FUNCTION_BLOCK PUBLIC FileSystemEntryCollection IMPLEMENTS I_FileSystemEntryCollection 
VAR
	entries : ARRAY[0..99] OF I_FileSystemEntry;
	currentIndex : INT := EMPTY;
	_nullEntry : NullEntry(Path:='');
END_VAR
VAR CONSTANT
	EMPTY : INT :=  -1;
END_VAR

METHOD Clear
VAR
	i : INT;
END_VAR
FOR i := 0 TO currentIndex DO
	entries[i] := 0;
END_FOR

THIS^.currentIndex := EMPTY;
END_METHOD

PROPERTY Count : UDINT
GET
Count := currentIndex + 1;
END_GET
END_PROPERTY

METHOD GetFirst : I_FileSystemEntry
IF NOT (Count > 0) THEN
	GetFirst := _nullEntry;
	RETURN;
END_IF

GetFirst := entries[0];
END_METHOD

METHOD GetNext : I_FileSystemEntry
VAR_INPUT
	Entry : I_FileSystemEntry;
END_VAR
VAR
	i : INT;
END_VAR
IF Count = 0 THEN
	GetNext := _nullEntry;
	RETURN;
END_IF

IF Entry = 0 THEN
	GetNext := GetFirst();
	RETURN;
END_IF

IF Entry = entries[currentIndex] THEN
	GetNext := _nullEntry;
	RETURN;
END_IF

FOR i := 0 TO currentIndex DO
	IF entries[i] = Entry THEN
		GetNext := entries[i+1];
		RETURN;
	END_IF
END_FOR

GetNext := _nullEntry;
END_METHOD

METHOD Insert
VAR_INPUT
	Entry : I_FileSystemEntry;
END_VAR
IF (currentIndex >= 99) THEN
	RETURN;
END_IF

currentIndex := currentIndex + 1;
entries[currentIndex] := Entry;
END_METHOD

END_FUNCTION_BLOCK

(* stored: Version 1.1.0.1, ProductVersion 3.1.4024.9
   POU FileSystemEntryCollection: Id {49c9c029-3eeb-4573-867b-19af0dafd403}, SpecialFunc None
   Method Clear: Id {a224ce7d-bcaf-423b-b0e7-f06a8769b3c5}
   Property Count: Id {e59573c1-3063-4ab4-8ae8-0e5af34953b5}
   Get Get: Id {3d15a0d4-e7a4-47c2-9929-06234fd411a7}
   Method GetFirst: Id {2b71e296-9901-4c08-a631-7758f9f4b506}
   Method GetNext: Id {67c41f2a-0b1a-43cb-bd0a-d6aac499ca99}
   Method Insert: Id {ba078abe-d739-48b8-8a39-755b79a391ec} *)
